// TIA Portal V19 export
TYPE "LAF_typeDevDiagNoOfDevices"
TITLE = Number of devices / Anzahl devices
// This data type contains the number of devices which have the respective status. / Struktur Anzahl devices PN device diag
// stored: Access Published
   STRUCT
      configured : UInt;   // - konfiguriert / Configured
      notPresent : UInt;   // - nicht vorhanden / Not present
      deactivated : UInt;   // - deaktiviert / Deactivated
      faulty : UInt;   // - gestört / Faulty
      problem : UInt;   // - Problem / Problem
   END_STRUCT;
END_TYPE
